// TIA Portal V20 export
// export: Created 2025-12-01T14:57:03.5259775Z, ExportSetting None, DisplayName Totally Integrated Automation Portal, DisplayVersion V20 Update 3, DisplayName TIA Portal Openness, DisplayVersion V20 Update 3, DisplayName TIA Portal Version Control Interface, DisplayVersion V20 Update 3, DisplayName STEP 7 Professional, DisplayVersion V20 Update 3, DisplayName STEP 7 Safety, DisplayVersion V20 Update 2, DisplayName WinCC Basic/Comfort/Advanced, DisplayVersion V20 Update 3, DisplayName WinCC Professional, DisplayVersion V20 Update 3, DisplayName WinCC Unified, DisplayVersion V20 Update 3
FUNCTION "FC701_JDT02ControlCOM" : Void   // FC701, LAD
TITLE = "ControlCOM" - Control de Comunicaciones
{ S7_Optimized_Access := 'FALSE' }
AUTHOR : TRACKING
NAME : 20150129
VERSION : 3.1
// - Contorol y valida el Enlace entre el PLC y el PC
// - Varible: EnlaceCP_OK
// stored: AutoNumber false, SetENOAutomatically false
   VAR_TEMP
      Temporal : Struct   // Temporal para el tratamiento de Result 01
         "0.0" : Bool;
         "0.1" : Bool;
         "0.2" : Bool;
         "0.3" : Bool;
         "0.4" : Bool;
         "0.5" : Bool;
         "0.6" : Bool;
         "0.7" : Bool;
         "1.0" : Bool;
         "1.1" : Bool;
         "1.2" : Bool;
         "1.3" : Bool;
         "1.4" : Bool;
         "1.5" : Bool;
         "1.6" : Bool;
         "1.7" : Bool;
         "2.0" : Bool;
         "2.1" : Bool;
         "2.2" : Bool;
         "2.3" : Bool;
         "2.4" : Bool;
         "2.5" : Bool;
         "2.6" : Bool;
         "2.7" : Bool;
         "3.0" : Bool;
         "3.1" : Bool;
         "3.2" : Bool;
         "3.4" : Bool;
         "3.5" : Bool;
         "3.6" : Bool;
         "3.7" : Bool;
      END_STRUCT;
      P_Temporal : DWord;
      TMPEnlace_OK : Bool;
   END_VAR
BEGIN

NETWORK
TITLE = Control del Enlace - Puerto 2001
// - Distribución  - Conexion  - Desconesion  - Final    ------------------------------------------------------------------------------------------------------   Control del Enlace - Distribución   --- Si hay que desconetar   --- Si esta conectado
      A     "DB701_JDT02StatusCOM".CNTRL_Reset;  // Si hay que desconectar
      O     "DB701_JDT02StatusCOM".RecJdT_Reset;
      O     "DB701_JDT02StatusCOM".EmiJdT_Reset;
      JC    DesConectar;

      A     "DB701_JDT02StatusCOM".EnlaceCP_OK;  // Si está conectado
      JC    Final;

      JU    Conectar;  // Hay que conectar

// ------------------------------------------------------------------------------------------------------
// Control del Enlace - Conexion
// --- Mirar si hay que activar Flanco
// --- Mirar si hay petición de conexion activa
// --- Llamada de Conexion
// --- Comprobación de la Conexion

Conectar:NOP   0;
      AN    "DB891_VariablesTCP".TCON_JdT_PLC_Busy_JDT02;
      AN    "DB891_VariablesTCP".TCON_JdT_PLC_Req_JDT02;
      AN    "DB891_VariablesTCP".TCON_JdT_PLC_Flanco_JDT02;
      =     "DB891_VariablesTCP".TCON_JdT_PLC_Flanco_JDT02;  // -- Activar flanco

      A     "DB891_VariablesTCP".TCON_JdT_PLC_Flanco_JDT02;
      AN    "DB891_VariablesTCP".TCON_JdT_PLC_Req_JDT02;
      S     "DB891_VariablesTCP".TCON_JdT_PLC_Req_JDT02;
      R     "DB891_VariablesTCP".TDISCON_JdT_PLC_Req_JDT02;  // -- Petición de Conexion Activa

      CALL  TCON, "DB896_TCON_JdT_PLC_JDT02"
      ( REQ     := "DB891_VariablesTCP".TCON_JdT_PLC_Flanco_JDT02,
        ID      := W#16#3,
        DONE    := "DB891_VariablesTCP".TCON_JdT_PLC_Done_JDT02,
        BUSY    := "DB891_VariablesTCP".TCON_JdT_PLC_Busy_JDT02,
        ERROR   := "DB891_VariablesTCP".TCON_JdT_PLC_Error_JDT02,
        STATUS  := "DB891_VariablesTCP".TCON_JdT_PLC_Status_JDT02,
        CONNECT := "DB700_JDTD02ConfigEnlace"
      );


      A     "DB891_VariablesTCP".TCON_JdT_PLC_Done_JDT02;  // -- Comprobacion de la Conexion
      R     "DB891_VariablesTCP".TCON_JdT_PLC_Req_JDT02;
      S     "DB701_JDT02StatusCOM".EnlaceCP_OK;

      A     "DB891_VariablesTCP".TCON_JdT_PLC_Error_JDT02;  // -- Error en conexion
      R     "DB891_VariablesTCP".TCON_JdT_PLC_Req_JDT02;

      A     "DB891_VariablesTCP".TCON_JdT_PLC_Req_JDT02;  // --- Control de Bloqueo
      AN    "DB891_VariablesTCP".TCON_JdT_PLC_Busy_JDT02;
      R     "DB891_VariablesTCP".TCON_JdT_PLC_Req_JDT02;

      JU    Final;  // Fin de la Conexión

// ------------------------------------------------------------------------------------------------------
// Control del Enlace - Desconexion
// --- Mirar si hay que activar Flanco
// --- Mirar si hay petición de desconexion activa
// --- Llamada de DesConexion
// --- Comprobación de la DesConexion

DesConectar:SET;
      R     "DB701_JDT02StatusCOM".EnlaceCP_OK;

      AN    "DB891_VariablesTCP".TDISCON_JdT_PLC_Busy_JDT02;
      AN    "DB891_VariablesTCP".TDISCON_JdT_PLC_Req_JDT02;
      AN    "DB891_VariablesTCP".TDISCON_JdT_PLC_Flanco_JDT02;
      =     "DB891_VariablesTCP".TDISCON_JdT_PLC_Flanco_JDT02;  // -- Activar Flanco


      A     "DB891_VariablesTCP".TDISCON_JdT_PLC_Flanco_JDT02;
      AN    "DB891_VariablesTCP".TDISCON_JdT_PLC_Req_JDT02;
      S     "DB891_VariablesTCP".TDISCON_JdT_PLC_Req_JDT02;
      R     "DB891_VariablesTCP".TCON_JdT_PLC_Req_JDT02;  // -- Petición de DesConexion Activa

      CALL  TDISCON, "DB897_TDISCON_JdT_PLC_JDT02"
      ( REQ    := "DB891_VariablesTCP".TDISCON_JdT_PLC_Flanco_JDT02,
        ID     := W#16#3,
        DONE   := "DB891_VariablesTCP".TDISCON_JdT_PLC_Done_JDT02,
        BUSY   := "DB891_VariablesTCP".TDISCON_JdT_PLC_Busy_JDT02,
        ERROR  := "DB891_VariablesTCP".TDISCON_JdT_PLC_Error_JDT02,
        STATUS := "DB891_VariablesTCP".TDISCON_JdT_PLC_Status_JDT02
      );



      A     "DB891_VariablesTCP".TDISCON_JdT_PLC_Done_JDT02;  // -- Comprobacion de la DesConexión
      R     "DB891_VariablesTCP".TDISCON_JdT_PLC_Req_JDT02;


      R     "DB701_JDT02StatusCOM".CNTRL_Reset;
      R     "DB701_JDT02StatusCOM".RecJdT_Reset;
      R     "DB701_JDT02StatusCOM".EmiJdT_Reset;

      A     "DB891_VariablesTCP".TDISCON_JdT_PLC_Error_JDT02;  // -- Error en la DesConexion
      R     "DB891_VariablesTCP".TDISCON_JdT_PLC_Req_JDT02;

      O(;
      L     "DB891_VariablesTCP".TDISCON_JdT_PLC_Status_JDT02;
      L     W#16#80A3;  //Se está intentando deshacer una conexión no existente
      ==I;
      );
      O(;
      L     "DB891_VariablesTCP".TDISCON_JdT_PLC_Status_JDT02;
      L     W#16#8086;  //El parámetro ID se encuentra en un rango no permitido
      ==I;
      );
      R     "DB891_VariablesTCP".TDISCON_JdT_PLC_Busy_JDT02;
      R     "DB891_VariablesTCP".TDISCON_JdT_PLC_Req_JDT02;
      R     "DB891_VariablesTCP".TDISCON_JdT_PLC_Flanco_JDT02;

      A     "DB891_VariablesTCP".TDISCON_JdT_PLC_Req_JDT02;  // --- Control de Bloqueo
      AN    "DB891_VariablesTCP".TDISCON_JdT_PLC_Busy_JDT02;
      R     "DB891_VariablesTCP".TDISCON_JdT_PLC_Req_JDT02;

      R     "DB701_JDT02StatusCOM".CNTRL_Reset;
      R     "DB701_JDT02StatusCOM".RecJdT_Reset;
      R     "DB701_JDT02StatusCOM".EmiJdT_Reset;

      JU    Final;  // Fin de la DesConexión

// ------------------------------------------------------------------------------------------------------
// Control del Enlace - Final

Final:NOP   0;


END_FUNCTION
